// Struckig
// Copyright (C) 2022 Stefan Besler

// This program is free software: you can redistribute it and/or modify
// it under the terms of the GNU General Public License as published by
// the Free Software Foundation, either version 3 of the License, or
// (at your option) any later version.

// This program is distributed in the hope that it will be useful,
// but WITHOUT ANY WARRANTY; without even the implied warranty of
// MERCHANTABILITY or FITNESS FOR A PARTICULAR PURPOSE.  See the
// GNU General Public License for more details.
//
// You should have received a copy of the GNU General Public License
// along with THIS PROGRAM.  IF NOT, see <http://www.gnu.org/licenses/>.
{attribute 'qualified_only'}
{attribute 'strict'}
TYPE INTERNAL ProfileDirection :
(
  Up,
  Down
);
END_TYPE

(* stored: Version 1.1.0.1
   DUT ProfileDirection: Id {2ff73edb-5bff-447c-9ade-9d123b5bb840} *)
